// TIA Portal V20 export
TYPE "LER_typeTwoWayActuatorInterlock"
// stored: Access Published
   STRUCT
      home : Bool;
      work : Bool;
   END_STRUCT;
END_TYPE
